FUNCTION TryConvert_DATE_TO_REAL : BOOL
VAR_INPUT
	in : DATE;
	out : REFERENCE TO REAL;
END_VAR

out := DATE_TO_REAL(in);
TryConvert_DATE_TO_REAL := TRUE;

END_FUNCTION

(* stored: Version 1.1.0.1, ProductVersion 3.1.4024.12
   POU TryConvert_DATE_TO_REAL: Id {04ef4155-eed7-475a-b712-2c9913c9b5a7}, SpecialFunc None *)
